IF I_bWebOn
THEN
	Q_sConvString:=	CONCAT(F_ToCHR(I_sStartZeichen),DINT_TO_STRING(I_diID));
	Q_sConvString:=	CONCAT(Q_sConvString,'.SYS.');
	Q_sConvString:=	CONCAT(Q_sConvString,INT_TO_STRING(1));
	Q_sConvString:=	CONCAT(Q_sConvString,'.WEBSERVER.');
	Q_sConvString:=	CONCAT(Q_sConvString,INT_TO_STRING(1));
	Q_sConvString:=	CONCAT(Q_sConvString,F_ToCHR(I_sEndZeichen));
ELSE
	Q_sConvString:=	CONCAT(F_ToCHR(I_sStartZeichen),DINT_TO_STRING(I_diID));
	Q_sConvString:=	CONCAT(Q_sConvString,'.SYS.');
	Q_sConvString:=	CONCAT(Q_sConvString,INT_TO_STRING(1));
	Q_sConvString:=	CONCAT(Q_sConvString,'.WEBSERVER.');
	Q_sConvString:=	CONCAT(Q_sConvString,INT_TO_STRING(0));
	Q_sConvString:=	CONCAT(Q_sConvString,F_ToCHR(I_sEndZeichen));
END_IF

END_FUNCTION_BLOCK

// ---- POUs/RS485_Hausbus_FB/CYD/fb_StringConvCYDWifi.TcPOU
(*======================================================================================================================================*)
(*fb_StringConvTB6F:	Zusammensetzen des Strings für 6Fach Bust Taster (LEDs und Hintergrundbeleuchtung und Reset)*)
(*
Date          	| Version    	| created under        	| Author          	| Remark *)
(*====================================================================================================================================================*)
(*05/05/2025   	| 1.00      		| TC3		  		| N.Kersting       | first release *)
(*06/05/2025   	| 1.01      		| TC3		  		| N.Kersting       | Externe LEDs Nachgerüstet *)
(*08/05/2025   	| 1.02      		| TC3		  		| N.Kersting       | Umschaltung ob Externe LEDs verwendet werden oder nicht *)
(*22/05/2025   	| 1.03      		| TC3		  		| N.Kersting       | Spezialversion für CYD *)
(*====================================================================================================================================================*)
FUNCTION_BLOCK fb_StringConvCYDWifi
VAR_INPUT
	I_diID				:DINT;							(* Device ID *)
	I_bWIFIOn			:BOOL;
	I_sStartZeichen		:BYTE := 16#FD;					(* Startzeichen Präfix *)
	I_sEndZeichen		:BYTE := 16#FE;					(* Endzeichen Suffix *)
END_VAR
VAR_OUTPUT
	Q_sConvString		:STRING(255);
END_VAR
VAR
END_VAR


IF I_bWIFIOn
THEN
	Q_sConvString:=	CONCAT(F_ToCHR(I_sStartZeichen),DINT_TO_STRING(I_diID));
	Q_sConvString:=	CONCAT(Q_sConvString,'.SYS.');
	Q_sConvString:=	CONCAT(Q_sConvString,INT_TO_STRING(1));
	Q_sConvString:=	CONCAT(Q_sConvString,'.WIFI.');
	Q_sConvString:=	CONCAT(Q_sConvString,INT_TO_STRING(1));
	Q_sConvString:=	CONCAT(Q_sConvString,F_ToCHR(I_sEndZeichen));
else
	Q_sConvString:=	CONCAT(F_ToCHR(I_sStartZeichen),DINT_TO_STRING(I_diID));
	Q_sConvString:=	CONCAT(Q_sConvString,'.SYS.');
	Q_sConvString:=	CONCAT(Q_sConvString,INT_TO_STRING(1));
	Q_sConvString:=	CONCAT(Q_sConvString,'.WIFI.');
	Q_sConvString:=	CONCAT(Q_sConvString,INT_TO_STRING(0));
	Q_sConvString:=	CONCAT(Q_sConvString,F_ToCHR(I_sEndZeichen));
END_IF

END_FUNCTION_BLOCK

// ---- POUs/RS485_Hausbus_FB/CYD/fb_StringConvCYDService.TcPOU
(*======================================================================================================================================*)
(*fb_StringConvTB6F:	Zusammensetzen des Strings für 6Fach Bust Taster (LEDs und Hintergrundbeleuchtung und Reset)*)
(*
Date          	| Version    	| created under        	| Author          	| Remark *)
(*====================================================================================================================================================*)
(*05/05/2025   	| 1.00      		| TC3		  		| N.Kersting       | first release *)
(*06/05/2025   	| 1.01      		| TC3		  		| N.Kersting       | Externe LEDs Nachgerüstet *)
(*08/05/2025   	| 1.02      		| TC3		  		| N.Kersting       | Umschaltung ob Externe LEDs verwendet werden oder nicht *)
(*22/05/2025   	| 1.03      		| TC3		  		| N.Kersting       | Spezialversion für CYD *)
(*====================================================================================================================================================*)
FUNCTION_BLOCK fb_StringConvCYDService
VAR_INPUT
	I_diID				:DINT;							(* Device ID *)
	I_bServiceOn		:BOOL;
	I_sStartZeichen		:BYTE := 16#FD;					(* Startzeichen Präfix *)
	I_sEndZeichen		:BYTE := 16#FE;					(* Endzeichen Suffix *)
END_VAR
VAR_OUTPUT
	Q_sConvString		:STRING(255);
END_VAR
VAR
END_VAR


IF I_bServiceOn
THEN
	Q_sConvString:=	CONCAT(F_ToCHR(I_sStartZeichen),DINT_TO_STRING(I_diID));
	Q_sConvString:=	CONCAT(Q_sConvString,'.SYS.');
	Q_sConvString:=	CONCAT(Q_sConvString,INT_TO_STRING(1));
	Q_sConvString:=	CONCAT(Q_sConvString,'.SERVICE.');
	Q_sConvString:=	CONCAT(Q_sConvString,INT_TO_STRING(1));
	Q_sConvString:=	CONCAT(Q_sConvString,F_ToCHR(I_sEndZeichen));
ELSE
	Q_sConvString:=	CONCAT(F_ToCHR(I_sStartZeichen),DINT_TO_STRING(I_diID));
	Q_sConvString:=	CONCAT(Q_sConvString,'.SYS.');
	Q_sConvString:=	CONCAT(Q_sConvString,INT_TO_STRING(1));
	Q_sConvString:=	CONCAT(Q_sConvString,'.SERVICE.');
	Q_sConvString:=	CONCAT(Q_sConvString,INT_TO_STRING(0));
	Q_sConvString:=	CONCAT(Q_sConvString,F_ToCHR(I_sEndZeichen));
END_IF

END_FUNCTION_BLOCK

// ---- POUs/RS485_Hausbus_FB/RS485 COM/fb_RS485ComCheck.TcPOU
(*======================================================================================================================================*)
(*fb_RS485ComCheck:	Einfacher Universal Ping Baustein um von allerlei Geräten von haus-bus.de Kommunikation zu Checken über RS485 
	In Diesem Fall ist es für einen Taster (BTN) bei einem Relais sollte es (OUT) sein*)
(*
Date          	| Version    	| created under        	| Author          	| Remark *)
(*====================================================================================================================================================*)
(*05/05/2025   	| 1.00      		| TC3		  		| N.Kersting       | first release *)
(*06/05/2025   	| 1.01      		| TC3		  		| N.Kersting       | Bugfix Timeouts werden besser ausgewertet *)
(*07/05/2025   	| 1.02      		| TC3		  		| N.Kersting       | Bug in Schritt 2 behoben (weiter, wenn nicht Busy) *)
(*09/05/2025   	| 1.03      		| TC3		  		| N.Kersting       | Counter für verbindungsversuche inkl. erneut senden *)
(*10/05/2025   	| 1.04      		| TC3		  		| N.Kersting       | Umrüstung Auf Externen Fifo  *)
(*12/05/2025   	| 1.05      		| TC3		  		| N.Kersting       | Verriegelung über I_bStart, damit nich gesendet werden kann wenn nicht Freigegeben  *)
(*14/05/2025   	| 1.06      		| TC3		  		| N.Kersting       | Ausgänge ergänzt für Done  *)
(*27/05/2025   	| 1.07      		| TC3		  		| N.Kersting       | Aufgeräumt und wesentlich bessere Auswertung Es wird nicht mehr auf Instanz ID geachtet beim receive  *)
(*====================================================================================================================================================*)
FUNCTION_BLOCK fb_RS485ComCheck
VAR_INPUT
	I_FifoID			:INT;
	I_bExecute			:BOOL;							(* Aktiviert den Baustein *)
	I_bStart			:BOOL;							(* Startet das Senden des Pings *)
	I_tPingIntervall	:TIME := T#5S;					(* Intervall Zeit wann die Kommunikation geprüft werden soll *)
	I_tPingTimeout		:TIME := T#2S;					(* Zeit, bis der Ping zurück gekommen sein muss *)
	I_diID				:DINT;							(* Device ID *)
	I_sPingSymbol		:STRING :='.BTN.';				(* Symbol, welches als Ping genutzt werden soll *)
	I_iInstID			:INT := 17;						(* Instanz ID  wird nur zum senden des Abfragebefehls verwendet! *)
	I_sStartZeichen		:BYTE := 16#FD;					(* Startzeichen Präfix *)
	I_sEndZeichen		:BYTE := 16#FE;					(* Endzeichen Suffix *)
	I_StringReceived	:STRING(255);					(* Empfangener String *)
	I_iMaxPingTry		:INT := 5;
END_VAR
VAR_OUTPUT
	Q_sSend				:STRING(255);
	Q_bBusy 			:BOOL;
	Q_bSendDone			:BOOL;
	Q_sState			:STRING;
	Q_bComOk			:BOOL;
	Q_bTimeout			:BOOL;
	Q_bError			:BOOL;
END_VAR
VAR
	sStringSend			:STRING;
	fbBusPingEvent		:fb_BusPingEvent;
	
	tonIntervall		:ton;
	tonTimeout			:ton;
	tonRecevieAutoReset	:ton;
	
	iStepReceive		:INT;
	iStep				:INT;
	icntComTry			:INT;
	iMaxComTry			:INT := 5;
	i					:INT;
	icntSymbole			:INT;
	
	bSend				:BOOL;
	bReceived			:BOOL;
	bCOMMem				:BOOL;
END_VAR

iMaxComTry :=	I_iMaxPingTry;

(* Intervall timer *)
tonIntervall(
	PT := I_tPingIntervall);
	
(* Timeout timer *)
tonTimeout(
	PT := I_tPingTimeout);
	
(* Ping String ertsllen *)
sStringSend:=	CONCAT(F_ToCHR(I_sStartZeichen),DINT_TO_STRING(I_diID));
sStringSend:=	CONCAT(sStringSend,I_sPingSymbol);
sStringSend:=	CONCAT(sStringSend,INT_TO_STRING(I_iInstID));
sStringSend:=	CONCAT(sStringSend,'.gSTATUS');
sStringSend:=	CONCAT(sStringSend,F_ToCHR(I_sEndZeichen));

IF NOT I_bExecute 
	AND NOT I_bStart
THEN
	Q_bComOk := FALSE;
	Q_bTimeout := FALSE;
	tonIntervall.IN := FALSE;
	tonTimeout.IN := FALSE;
	sStringSend:= '';
	bSend := FALSE;
	iStep := 0;
ELSE
	ac01_Send();
END_IF

ACTION ac01_Send:
(* Sende Schrittkette *)
			
CASE iStep OF
(*=========================================================*)	
0:	Q_sState := ' INIT';
	tonIntervall.IN := FALSE;
	tonTimeout.IN := FALSE;
	bCOMMem := FALSE;
	bSend := FALSE;
	Q_bBusy := FALSE;
	Q_sSend := '';
	
	IF I_bExecute
		AND I_bStart
	THEN
		Q_bSendDone := FALSE;
		Q_bBusy := TRUE;
		iStep := iStep +1;
	ELSIF
		NOT I_bExecute
	THEN
		iStep := 10;
	END_IF

(*=========================================================*)	
1:	Q_sState := 'Starte Sendebefehl';
	
	IF GVL_RS485FiFoSend.bSendDoneFiFo[I_FifoID]
	THEN
		tonTimeout.IN := TRUE;
		Q_sSend := sStringSend;
	END_IF
	IF NOT GVL_RS485FiFoSend.bSendDoneFiFo[I_FifoID]
	THEN
		tonTimeout.IN := FALSE;
		iStep := iStep +1;
	ELSIF
		tonTimeout.Q
	THEN
		tonTimeout.IN := FALSE;
		Q_sState := 'Timeout Send Busy';
		iStep := -1;
	END_IF
	
(*=========================================================*)	
2:	Q_sState := 'Auswertung Senden';
	bSend := FALSE;	
	tonTimeout.IN := TRUE;
	
	IF GVL_RS485FiFoSend.bSendDoneFiFo[I_FifoID]
	THEN
		Q_sSend := '';
		Q_bSendDone := TRUE;
		tonTimeout.IN := FALSE;
		iStep := iStep +1;
	ELSIF
		tonTimeout.Q
	THEN
		Q_sState := 'Timeout Send Done';
		iStep := -2;
	END_IF
		
(*=========================================================*)	
3:	Q_sState := 'Warte auf Empfang';
	tonTimeout.IN := TRUE;
	
	IF tonTimeout.Q
	THEN
		(* Kommunikations versuche *)
		IF icntComTry <iMaxComTry
		THEN
			icntComTry := icntComTry +1;
			iStep := 5;				(* Erneut Senden *)
		ELSE
			Q_sState := 'Timeout kein Ping Empfangen';
			Q_bComOk := FALSE;
			Q_bTimeout := TRUE;
			iStep := -4;	(* Erneut Empfangen *)
		END_IF
	ELSE
		
		IF	bCOMMem
		THEN
			bCOMMem := FALSE;
			iStep := iStep+1;		(* Telegram erhalten *)
		END_IF
	END_IF
	
(*=========================================================*)	
4:	Q_sState := 'Ping Empfangen, Warte auf Intervall';
	tonIntervall.IN := TRUE;
	Q_bComOk := TRUE;
	Q_bTimeout := FALSE;
	
	IF tonIntervall.Q
		AND I_bStart
	THEN
		icntComTry := 0;	(* Wenn die Verbindung wieder da ist dürfen die Versuche gelöscht werden *)
		iStep := 0;
	END_IF

(*=========================================================*)	
5:	Q_sState := 'Ping nicht Empfangen, Warte auf Intervall';
	tonIntervall.IN := TRUE;
	
	IF tonIntervall.Q
		AND I_bStart
	THEN
		iStep := 0;
	END_IF

(*=========================================================*)	
10:	Q_sState := 'Warten Auf Automatischen Ping vom Taster';
	tonIntervall.IN := TRUE;
	
	IF tonIntervall.Q
		AND I_bStart
	THEN
		Q_bComOk := FALSE;
		iStep := 0;
	ELSE
		IF bCOMMem
		THEN
			tonIntervall.IN := FALSE;
			Q_bComOk := TRUE;
			iStep := 0;
		END_IF
	END_IF	
ELSE
	tonIntervall.IN := TRUE;
	tonTimeout.IN := FALSE;
	Q_bComOk := FALSE;
	bSend := FALSE;
	Q_bBusy := FALSE;
	icntComTry := 0;
	Q_sSend := '';
	
	IF tonIntervall.Q
		AND I_bStart
	THEN
		iStep := 0;
	END_IF
END_CASE

fbBusPingEvent(
	I_bReset := 			FALSE,
	I_sID:= 				DINT_TO_STRING(I_diID ),
	I_sReceivedString:= 	I_StringReceived, 
	Q_bOut=> 				);
	
IF iStep > 0
	AND fbBusPingEvent.Q_bOut
THEN
	bCOMMem := TRUE;
END_IF

(*	
IF I_bTasterMode
THEN
	icntSymbole := 0;
	(* Durchgehend Checken ob Ping kommt *)
	FOR i := 1 TO 6 BY 1 DO 
		
			
		IF fbBusPingEvent[i].Q_bOut
		THEN
			icntSymbole := icntSymbole +1;
		END_IF
	END_FOR
	
	IF iStep > 0
		AND icntSymbole >0
	THEN
		bCOMMem := TRUE;
	END_IF
ELSE
	(* Nur nach der einen ID Gucken *)
	fbBusPingEvent[1](
		I_bReset := 			FALSE,
		I_sID:= 				DINT_TO_STRING(I_diID ), 
		I_sReceivedString:= 	I_StringReceived, 
		Q_bOut=> 				);
		
	IF iStep > 0
		AND fbBusPingEvent[1].Q_bOut
	THEN
		bCOMMem := TRUE;
	END_IF
END_IF
*)
END_ACTION

END_FUNCTION_BLOCK

// ---- GlobalTextList.TcGTLO
TEXTLIST GlobalTextList
  573 = '%s'
  382 = 'BG LEDs: %s'
  258 = 'BTN1'
  576 = 'BTN1 %s'
  715 = 'BTN1Ext'
  23 = 'BTN2'
  297 = 'BTN2 '
  965 = 'BTN2 %s '
  554 = 'BTN2Ext'
  479 = 'BTN3'
  188 = 'BTN3 %s'
  737 = 'BTN3Ext'
  989 = 'BTN4'
  390 = 'BTN4 %s'
  345 = 'BTN4Ext'
  308 = 'BTN5'
  533 = 'BTN5 %s'
  511 = 'BTN5Ext'
  943 = 'BTN6'
  202 = 'BTN6 %s'
  907 = 'BTN6Ext'
  595 = 'BTN7'
  680 = 'BTN7 %s'
  941 = 'BTN8'
  988 = 'BTN8 %s'
  450 = 'Bus'
  700 = 'Bus Auslastung'
  874 = 'Bus Ok'
  355 = 'Busbelastungstest'
  902 = 'Busy'
  187 = 'COM'
  634 = 'Count %s '
  330 = 'CYD'
  1529 = 'Display: %s\nBeleuchtung'
  323 = 'Done'
  235 = 'Error'
  325 = "Externe E/A's"
  546 = 'Externe EA'
  790 = 'FiFo Master'
  587 = 'Gefundene Ids'
  29 = 'Hintergrund LEDs: %s'
  896 = 'Hintergrund: %s'
  246 = 'Humi: %s p'
  180 = "Interne E/A's"
  872 = 'Interne Eeingänge '
  925 = 'Interne Eingänge '
  921 = 'Lum: %s p'
  192 = 'Manuell'
  356 = 'R1'
  892 = 'R10'
  223 = 'R11'
  245 = 'R12'
  593 = 'R13'
  117 = 'R14'
  996 = 'R15'
  327 = 'R16'
  233 = 'R2'
  713 = 'R3'
  132 = 'R4'
  769 = 'R5'
  317 = 'R6'
  716 = 'R7'
  350 = 'R8'
  333 = 'R9'
  663 = 'Relais'
  267 = 'Relais '
  292 = 'Reset'
  342 = 'Row %s '
  289 = 'RX: %s'
  963 = 'Scan'
  743 = 'Senden'
  846 = 'Service Seite'
  458 = 'ServiceMode'
  172 = 'Startup\nDone'
  38 = 'Startup\nError'
  25 = 'Startup :%s '
  789 = 'State :%s '
  93 = 'Taster'
  696 = 'Temp: %s °C'
  495 = 'TX %s'
  18 = 'TX: %s'
  58 = 'Visu Service Mode'
  217 = 'WebServer'
  932 = 'Wifi'
END_TEXTLIST

// ---- VISUs/HausBus_RS485/BusCYD6F_Frame.TcVIS
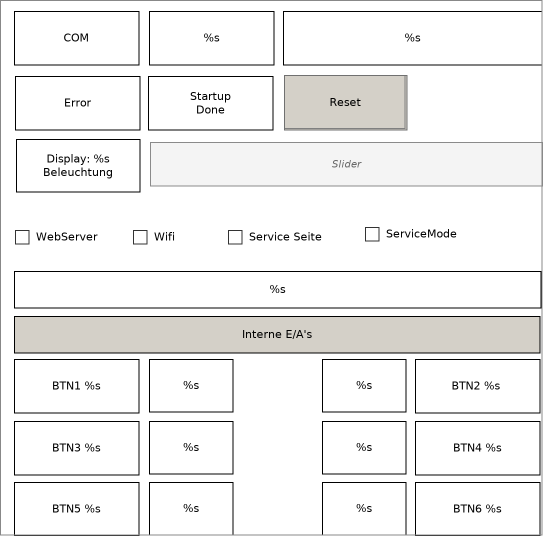
VISUALIZATION BusCYD6F_Frame  // 543x536
VAR_IN_OUT
	stBusTaster6F_Input		:ST_BusCYD6F_Input;
	stBusTaster6F_Output	:ST_BusTaster6F_Output;
	stBusTaster6F_Cnt		:ST_BusTaster6F_Cnt;
END_VAR
    Rectangle (14,11 125x54), "COM", colour toggle: stBusTaster6F_Output.bCOM
    Rectangle (14,359 125x54), "BTN1 %s", text variable: stBusTaster6F_Cnt.dwCntButtons[1], colour toggle: stBusTaster6F_Output.bButtons[1]
    Rectangle (149,11 125x54), "%s", text variable: stBusTaster6F_Input.diID
    Rectangle (283,11 259x54), "%s", text variable: stBusTaster6F_Input.sName
    Rectangle (415,359 125x54), "BTN2 %s", text variable: stBusTaster6F_Cnt.dwCntButtons[2], colour toggle: stBusTaster6F_Output.bButtons[2]
    Rectangle (14,421 125x54), "BTN3 %s", text variable: stBusTaster6F_Cnt.dwCntButtons[3], colour toggle: stBusTaster6F_Output.bButtons[3]
    Rectangle (415,421 125x54), "BTN4 %s", text variable: stBusTaster6F_Cnt.dwCntButtons[4], colour toggle: stBusTaster6F_Output.bButtons[4]
    Rectangle (14,482 125x54), "BTN5 %s", text variable: stBusTaster6F_Cnt.dwCntButtons[5], colour toggle: stBusTaster6F_Output.bButtons[5]
    Rectangle (415,482 125x54), "BTN6 %s", text variable: stBusTaster6F_Cnt.dwCntButtons[6], colour toggle: stBusTaster6F_Output.bButtons[6]
    Rectangle (149,359 84x53), "%s", text variable: stBusTaster6F_Input.iLED[1]
        OnMouseDown: write the text variable via VisuDialogs.Numpad, min 0, max 100
    Rectangle (322,359 84x53), "%s", text variable: stBusTaster6F_Input.iLED[2]
        OnMouseDown: write the text variable via VisuDialogs.Numpad, min 0, max 100
    Rectangle (149,421 84x53), "%s", text variable: stBusTaster6F_Input.iLED[3]
        OnMouseDown: write the text variable via VisuDialogs.Numpad, min 0, max 100
    Rectangle (322,421 84x53), "%s", text variable: stBusTaster6F_Input.iLED[4]
        OnMouseDown: write the text variable via VisuDialogs.Numpad, min 0, max 100
    Rectangle (149,482 84x53), "%s", text variable: stBusTaster6F_Input.iLED[5]
        OnMouseDown: write the text variable via VisuDialogs.Numpad, min 0, max 100
    Rectangle (322,482 84x53), "%s", text variable: stBusTaster6F_Input.iLED[6]
        OnMouseDown: write the text variable via VisuDialogs.Numpad, min 0, max 100
    Button (284,75 123x55), "Reset"
        tap stBusTaster6F_Input.bReset
    Rectangle (15,76 125x54), "Error", colour toggle: stBusTaster6F_Output.bError
    Rectangle (14,271 527x37), "%s", text variable: stBusTaster6F_Output.sState
    Rectangle (148,76 125x54), "Startup Done", colour toggle: stBusTaster6F_Output.bStartupDone
    Rectangle (16,139 124x53), "Display: %s Beleuchtung", text variable: stBusTaster6F_Input.iLEDBg
        OnMouseDown: write the text variable via VisuDialogs.Numpad, min 0, max 100
    Rectangle (14,316 526x37), "Interne E/A's"
    Slider (150,142 393x44), variable: stBusTaster6F_Input.iLEDBg, scale 0..100
    Checkbox (363,206 178x56), "ServiceMode", variable: stBusTaster6F_Input.bServiceMode
    Checkbox (13,213 121x48), "WebServer", variable: stBusTaster6F_Input.bWebServer, invisible if: not stBusTaster6F_Input.bServiceMode
    Checkbox (131,213 85x48), "Wifi", variable: stBusTaster6F_Input.bWifi, invisible if: not stBusTaster6F_Input.bServiceMode
    Checkbox (226,213 119x48), "Service Seite", variable: stBusTaster6F_Input.bService, invisible if: not stBusTaster6F_Input.bServiceMode
END_VISUALIZATION

// ---- VISUs/HausBus_RS485/BusRelais16F_Frame.TcVIS
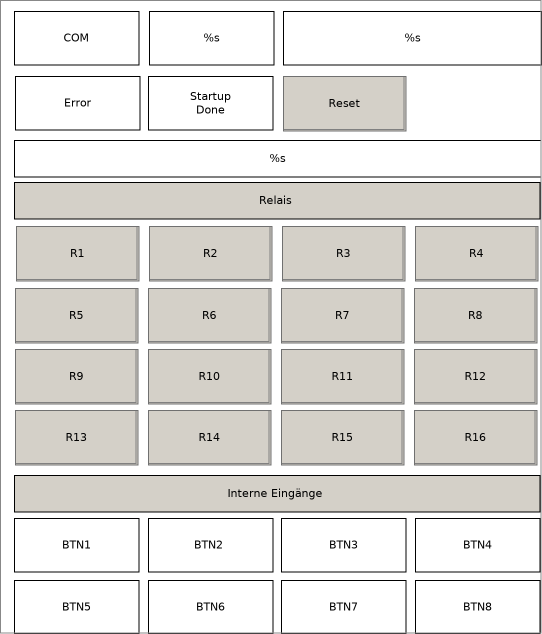
VISUALIZATION BusRelais16F_Frame  // 542x634
VAR_IN_OUT
	ST_BusRelais16F_Input		:ST_BusRelais16F_Input;
	ST_BusRelais16F_Output		:ST_BusRelais16F_Output;
	ST_BusRelais16F_Cnt			:ST_BusRelais16F_Cnt;
END_VAR
    Rectangle (14,11 125x54), "COM", colour toggle: ST_BusRelais16F_Output.bCOM
    Rectangle (14,518 125x54), "BTN1", colour toggle: ST_BusRelais16F_Output.bInputs[1]
    Rectangle (149,11 125x54), "%s", text variable: ST_BusRelais16F_Input.diID
    Rectangle (283,11 259x54), "%s", text variable: ST_BusRelais16F_Input.sName
    Rectangle (148,518 125x54), "BTN2", colour toggle: ST_BusRelais16F_Output.bInputs[2]
    Rectangle (281,518 125x54), "BTN3", colour toggle: ST_BusRelais16F_Output.bInputs[3]
    Rectangle (415,518 125x54), "BTN4", colour toggle: ST_BusRelais16F_Output.bInputs[4]
    Rectangle (14,580 125x54), "BTN5", colour toggle: ST_BusRelais16F_Output.bInputs[5]
    Rectangle (148,580 125x54), "BTN6", colour toggle: ST_BusRelais16F_Output.bInputs[6]
    Button (283,76 123x55), "Reset"
        tap ST_BusRelais16F_Input.bReset
    Rectangle (15,76 125x54), "Error", colour toggle: ST_BusRelais16F_Output.bError
    Rectangle (14,140 527x37), "%s", text variable: ST_BusRelais16F_Output.sState
    Rectangle (148,76 125x54), "Startup Done", colour toggle: ST_BusRelais16F_Output.bStartupDone
    Rectangle (14,475 526x37), "Interne Eingänge"
    Rectangle (281,580 125x54), "BTN7", colour toggle: ST_BusRelais16F_Output.bInputs[7]
    Rectangle (415,580 125x54), "BTN8", colour toggle: ST_BusRelais16F_Output.bInputs[8]
    Button (16,226 123x55), "R1"
        toggle ST_BusRelais16F_Input.bOut[1]
    Rectangle (14,182 526x37), "Relais"
    Button (149,226 123x55), "R2"
        toggle ST_BusRelais16F_Input.bOut[2]
    Button (282,226 123x55), "R3"
        toggle ST_BusRelais16F_Input.bOut[3]
    Button (415,226 123x55), "R4"
        toggle ST_BusRelais16F_Input.bOut[4]
    Button (15,288 123x55), "R5"
        toggle ST_BusRelais16F_Input.bOut[5]
    Button (148,288 123x55), "R6"
        toggle ST_BusRelais16F_Input.bOut[6]
    Button (281,288 123x55), "R7"
        toggle ST_BusRelais16F_Input.bOut[7]
    Button (414,288 123x55), "R8"
        toggle ST_BusRelais16F_Input.bOut[8]
    Button (15,349 123x55), "R9"
        toggle ST_BusRelais16F_Input.bOut[9]
    Button (148,349 123x55), "R10"
        toggle ST_BusRelais16F_Input.bOut[10]
    Button (281,349 123x55), "R11"
        toggle ST_BusRelais16F_Input.bOut[11]
    Button (414,349 123x55), "R12"
        toggle ST_BusRelais16F_Input.bOut[12]
    Button (15,410 123x55), "R13"
        toggle ST_BusRelais16F_Input.bOut[13]
    Button (148,410 123x55), "R14"
        toggle ST_BusRelais16F_Input.bOut[14]
    Button (281,410 123x55), "R15"
        toggle ST_BusRelais16F_Input.bOut[15]
    Button (414,410 123x55), "R16"
        toggle ST_BusRelais16F_Input.bOut[16]
END_VISUALIZATION

// ---- VISUs/HausBus_RS485/BusRS485Master_Frame.TcVIS
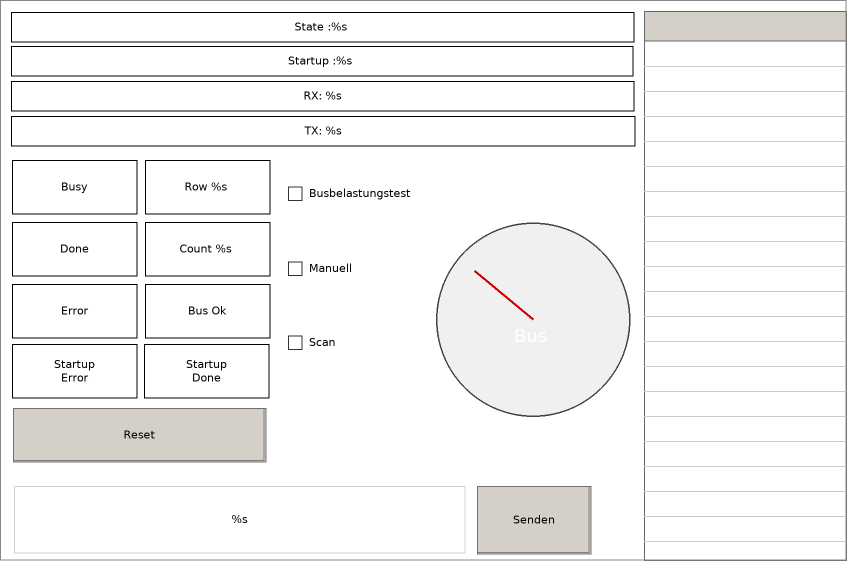
VISUALIZATION BusRS485Master_Frame  // 847x561
VAR_IN_OUT	
	(* für RS485 FiFo Master *)
	bBusBelastungstest		:BOOL;
	bReset					:BOOL;
	bSenden					:BOOL;
	sSenden					:STRING(255);
	bManuell				:BOOL;
	bIDScan					:BOOL;
	
	diScanIds				:ARRAY[1..cMaxScanIDs] OF DINT;
	stFiFoMasterState		:ST_FiFoMaster_State;
	stRS48StartupState		:ST_RS485Startup_State;
END_VAR
    Meter360 (436,202 194x235), value: stFiFoMasterState.lrBusAuslastung, style: Meter-Meter360-Gray, scale format: %.1f, scale 0..350
    Rectangle (11,81 623x30), "RX: %s", text variable: stFiFoMasterState.sReceiveString
    Checkbox (286,156 254x75), "Busbelastungstest", variable: bBusBelastungstest
    Rectangle (11,116 624x30), "TX: %s", text variable: stFiFoMasterState.sSendString
    Rectangle (11,12 623x30), "State :%s", text variable: stFiFoMasterState.sState
    Rectangle (12,160 125x54), "Busy", colour toggle: stFiFoMasterState.bBusy
    Rectangle (12,222 125x54), "Done", colour toggle: stFiFoMasterState.bDone
    Rectangle (12,284 125x54), "Error", colour toggle: stFiFoMasterState.bError
    Rectangle (145,160 125x54), "Row %s", text variable: stFiFoMasterState.iFiFoRow
    Rectangle (145,222 125x54), "Count %s", text variable: stFiFoMasterState.iFiFoCount
    Button (13,408 253x54), "Reset"
        tap bReset
    Label (456,321 150x30), "Bus"
    Rectangle (11,46 622x30), "Startup :%s", text variable: stRS48StartupState.sStartupState
    Rectangle (145,284 125x54), "Bus Ok", colour toggle: stRS48StartupState.bBusOk
    Rectangle (144,344 125x54), "Startup Done", colour toggle: stRS48StartupState.bStartupDone
    Rectangle (12,344 125x54), "Startup Error", colour toggle: stRS48StartupState.bStartupError
    Textfield (14,486 451x67), "%s", text variable: sSenden
        OnMouseDown: write the text variable via Edit
    Button (477,486 114x68), "Senden"
        tap bSenden
    Checkbox (286,231 138x75), "Manuell", variable: bManuell
    Checkbox (286,305 138x75), "Scan", variable: bIDScan, invisible if: not bManuell
    Table (644,11 203x550), data array: diScanIds
        p3854506369: diScanIds[INDEX]
        p2232123230: Gefundene Ids
END_VISUALIZATION

// ---- VISUs/HausBus_RS485/BusTatster6F_Frame.TcVIS
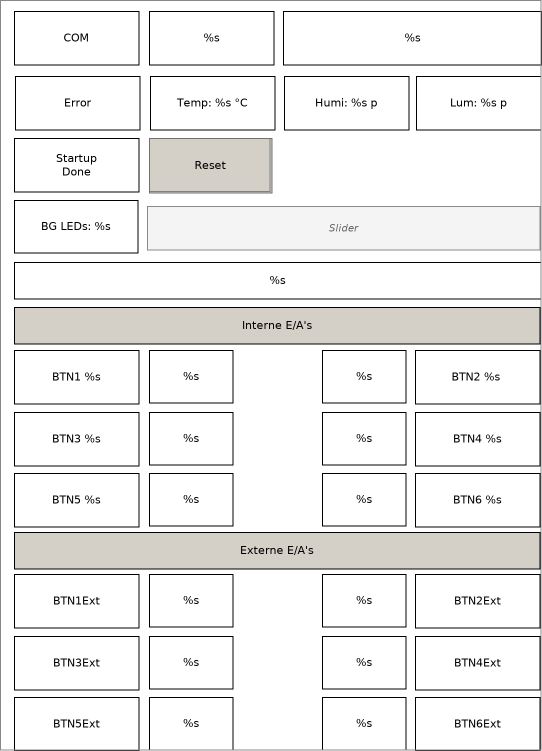
VISUALIZATION BusTatster6F_Frame  // 542x751
VAR_IN_OUT
	stBusTaster6F_Input		:ST_BusTaster6F_Input;
	stBusTaster6F_Output	:ST_BusTaster6F_Output;
	stBusTaster6F_Cnt		:ST_BusTaster6F_Cnt;
END_VAR
    Rectangle (14,11 125x54), "COM", colour toggle: stBusTaster6F_Output.bCOM
    Rectangle (14,350 125x54), "BTN1 %s", text variable: stBusTaster6F_Cnt.dwCntButtons[1], colour toggle: stBusTaster6F_Output.bButtons[1]
    Rectangle (149,11 125x54), "%s", text variable: stBusTaster6F_Input.diID
    Rectangle (283,11 259x54), "%s", text variable: stBusTaster6F_Input.sName
    Rectangle (415,350 125x54), "BTN2 %s", text variable: stBusTaster6F_Cnt.dwCntButtons[2], colour toggle: stBusTaster6F_Output.bButtons[2]
    Rectangle (14,412 125x54), "BTN3 %s", text variable: stBusTaster6F_Cnt.dwCntButtons[3], colour toggle: stBusTaster6F_Output.bButtons[3]
    Rectangle (415,412 125x54), "BTN4 %s", text variable: stBusTaster6F_Cnt.dwCntButtons[4], colour toggle: stBusTaster6F_Output.bButtons[4]
    Rectangle (14,473 125x54), "BTN5 %s", text variable: stBusTaster6F_Cnt.dwCntButtons[5], colour toggle: stBusTaster6F_Output.bButtons[5]
    Rectangle (415,473 125x54), "BTN6 %s", text variable: stBusTaster6F_Cnt.dwCntButtons[6], colour toggle: stBusTaster6F_Output.bButtons[6]
    Rectangle (149,350 84x53), "%s", text variable: stBusTaster6F_Input.iLED[1]
        OnMouseDown: write the text variable via VisuDialogs.Numpad, min 0, max 100
    Rectangle (322,350 84x53), "%s", text variable: stBusTaster6F_Input.iLED[2]
        OnMouseDown: write the text variable via VisuDialogs.Numpad, min 0, max 100
    Rectangle (149,412 84x53), "%s", text variable: stBusTaster6F_Input.iLED[3]
        OnMouseDown: write the text variable via VisuDialogs.Numpad, min 0, max 100
    Rectangle (322,412 84x53), "%s", text variable: stBusTaster6F_Input.iLED[4]
        OnMouseDown: write the text variable via VisuDialogs.Numpad, min 0, max 100
    Rectangle (149,473 84x53), "%s", text variable: stBusTaster6F_Input.iLED[5]
        OnMouseDown: write the text variable via VisuDialogs.Numpad, min 0, max 100
    Rectangle (322,473 84x53), "%s", text variable: stBusTaster6F_Input.iLED[6]
        OnMouseDown: write the text variable via VisuDialogs.Numpad, min 0, max 100
    Button (149,138 123x55), "Reset"
        tap stBusTaster6F_Input.bReset
    Rectangle (15,76 125x54), "Error", colour toggle: stBusTaster6F_Output.bError
    Rectangle (150,76 125x54), "Temp: %s °C", text variable: stBusTaster6F_Output.lrTemp
    Rectangle (284,76 125x54), "Humi: %s p", text variable: stBusTaster6F_Output.lrRhd
    Rectangle (416,76 125x54), "Lum: %s p", text variable: stBusTaster6F_Output.lrBrs
    Rectangle (14,262 527x37), "%s", text variable: stBusTaster6F_Output.sState
    Rectangle (14,138 125x54), "Startup Done", colour toggle: stBusTaster6F_Output.bStartupDone
    Rectangle (14,200 124x53), "BG LEDs: %s", text variable: stBusTaster6F_Input.iLEDBg
        OnMouseDown: write the text variable via VisuDialogs.Numpad, min 0, max 100
    Rectangle (14,574 125x54), "BTN1Ext", colour toggle: stBusTaster6F_Output.bButtonsExt[1]
    Rectangle (415,574 125x54), "BTN2Ext", colour toggle: stBusTaster6F_Output.bButtonsExt[2]
    Rectangle (14,636 125x54), "BTN3Ext", colour toggle: stBusTaster6F_Output.bButtonsExt[3]
    Rectangle (415,636 125x54), "BTN4Ext", colour toggle: stBusTaster6F_Output.bButtonsExt[4]
    Rectangle (14,697 125x54), "BTN5Ext", colour toggle: stBusTaster6F_Output.bButtonsExt[5]
    Rectangle (415,697 125x54), "BTN6Ext", colour toggle: stBusTaster6F_Output.bButtonsExt[6]
    Rectangle (149,574 84x53), "%s", text variable: stBusTaster6F_Input.iLEDExt[1]
        OnMouseDown: write the text variable via VisuDialogs.Numpad, min 0, max 100
    Rectangle (322,574 84x53), "%s", text variable: stBusTaster6F_Input.iLEDExt[2]
        OnMouseDown: write the text variable via VisuDialogs.Numpad, min 0, max 100
    Rectangle (149,636 84x53), "%s", text variable: stBusTaster6F_Input.iLEDExt[3]
        OnMouseDown: write the text variable via VisuDialogs.Numpad, min 0, max 100
    Rectangle (322,636 84x53), "%s", text variable: stBusTaster6F_Input.iLEDExt[4]
        OnMouseDown: write the text variable via VisuDialogs.Numpad, min 0, max 100
    Rectangle (149,697 84x53), "%s", text variable: stBusTaster6F_Input.iLEDExt[5]
        OnMouseDown: write the text variable via VisuDialogs.Numpad, min 0, max 100
    Rectangle (322,697 84x53), "%s", text variable: stBusTaster6F_Input.iLEDExt[6]
        OnMouseDown: write the text variable via VisuDialogs.Numpad, min 0, max 100
    Rectangle (14,532 526x37), "Externe E/A's"
    Rectangle (14,307 526x37), "Interne E/A's"
    Slider (147,206 393x44), variable: stBusTaster6F_Input.iLEDBg, scale 0..100
END_VISUALIZATION

// ---- VISUs/HausBus_RS485/RS485HB_ServiceVISU.TcVIS
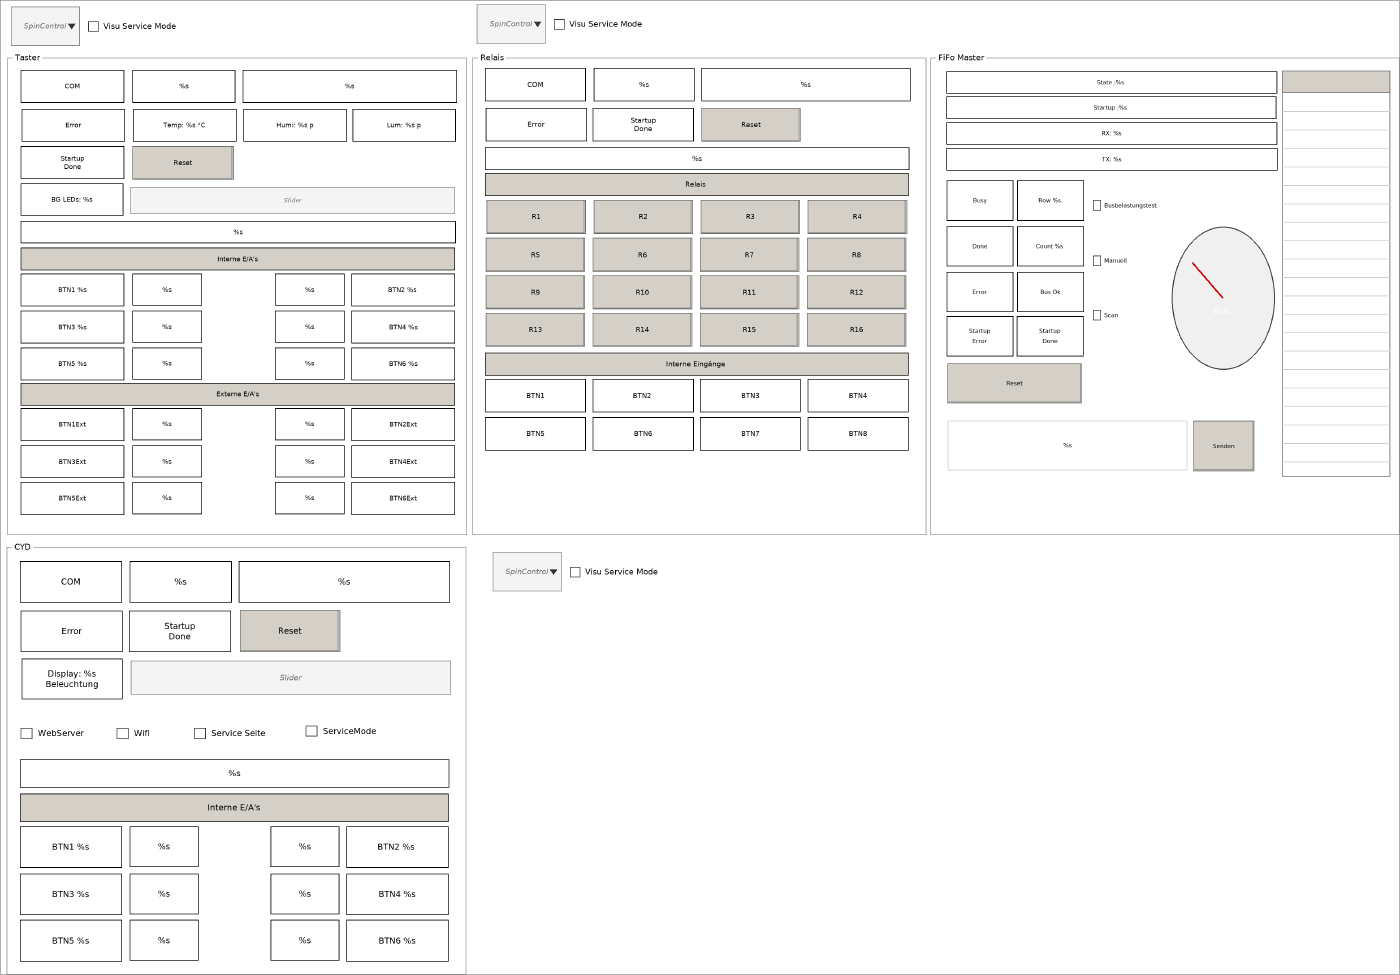
VISUALIZATION RS485HB_ServiceVISU  // 1938x1351
    SpinControl (15,9 95x54), variable: GVL_ServiceVisu.iDeviceTasterVisu
        p651134158: cMaxBusTaster
    Checkbox (120,7 181x59), "Visu Service Mode", variable: GVL_ServiceVisu.bTasterServiceAktiv[GVL_ServiceVisu.iDeviceTasterVisu]
    SpinControl (660,6 95x54), variable: GVL_ServiceVisu.iDeviceRelaisVisu
        p576042468: cMaxBusTaster+1
        p651134158: cMaxBusRelais +cMaxBusTaster +1
    Checkbox (765,4 181x59), "Visu Service Mode", variable: GVL_ServiceVisu.bRelaisServiceAktiv[GVL_ServiceVisu.iDeviceRelaisVisu]
    GroupBox (654,72 628x669), "Relais"
        Frame (2,13 604x539)
            shows BusRelais16F_Frame(ST_BusRelais16F_Input := GVL_ServiceVisu.stRelaisService[GVL_ServiceVisu.iDeviceRelaisVisu], ST_BusRelais16F_Output := fbRelaisHB16F[GVL_ServiceVisu.iDeviceRelaisVisu].Q_stOutput, ST_BusRelais16F_Cnt := fbRelaisHB16F[GVL_ServiceVisu.iDeviceRelaisVisu].Q_stCnt)
    GroupBox (10,72 636x669), "Taster"
        Frame (3,16 619x625)
            shows BusTatster6F_Frame(stBusTaster6F_Input := GVL_ServiceVisu.stTasterService[GVL_ServiceVisu.iDeviceTasterVisu], stBusTaster6F_Output := fbTasterHB6F[GVL_ServiceVisu.iDeviceTasterVisu].Q_stOutput, stBusTaster6F_Cnt := fbTasterHB6F[GVL_ServiceVisu.iDeviceTasterVisu].Q_stCnt)
    GroupBox (1288,72 650x669), "FiFo Master"
        Frame (14,15 622x573)
            shows BusRS485Master_Frame(bBusBelastungstest := RS485_COM_PRG.fbRS485SendCmdFiFo.I_bBusBelastungstest, bReset := RS485_COM_PRG.fbRS485SendCmdFiFo.I_bReset, bSenden := RS485_COM_PRG.fbRS485SendCmdFiFo.I_bSendManuell, sSenden := RS485_COM_PRG.fbRS485SendCmdFiFo.I_sSendCmdManuell, bManuell := RS485_COM_PRG.fbRS485SendCmdFiFo.I_bManuellMode, bIDScan := RS485_COM_PRG.fbRS485SendCmdFiFo.I_bSearchMode, diScanIds := RS485_COM_PRG.fbRS485SendCmdFiFo.fbRS485Search.Q_sIDList, stFiFoMasterState := RS485_COM_PRG.fbRS485SendCmdFiFo.Q_stStates, stRS48StartupState := RS485_COM_PRG.fbRS485Startup.Q_stStates)
            shows BusRS485Master_Frame()
    GroupBox (9,750 636x601), "CYD"
        Frame (3,16 612x566)
            shows BusCYD6F_Frame(stBusTaster6F_Input := GVL_ServiceVisu.stCYDService[GVL_ServiceVisu.iDeviceCYDVisu], stBusTaster6F_Output := fbCYDHB6F[GVL_ServiceVisu.iDeviceCYDVisu].Q_stOutput, stBusTaster6F_Cnt := fbCYDHB6F[GVL_ServiceVisu.iDeviceCYDVisu].Q_stCnt)
    SpinControl (682,765 95x54), variable: GVL_ServiceVisu.iDeviceCYDVisu
        p576042468: cMaxBusRelais +cMaxBusTaster +2
        p651134158: cMaxCYD+cMaxBusRelais +cMaxBusTaster +1
    Checkbox (787,763 181x59), "Visu Service Mode", variable: GVL_ServiceVisu.bCYDServiceAktiv[GVL_ServiceVisu.iDeviceCYDVisu]
END_VISUALIZATION
